TYPE ST_ViciControl :
STRUCT
	sViciReply			: STRING;
	iReqPos				: INT;
	xDirection			:BOOL;
	iAddress				:INT;
END_STRUCT
END_TYPE

(* stored: Version 1.1.0.1, ProductVersion 3.1.4020.6
   DUT ST_ViciControl: Id {3dbe2ab7-c9fe-4a0a-8fa6-39ab515d681c} *)
